// Mitsubishi GX Works2 project: PLC 특수기능 (BKRST)   PLC: Q03UDV

PROGRAM MAIN
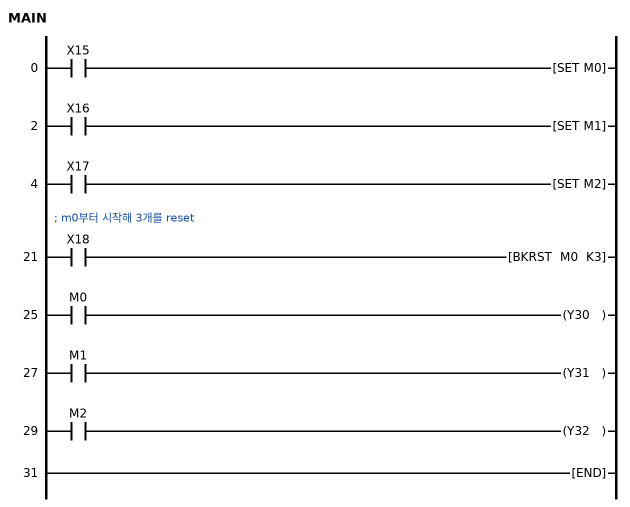
0     LD      X15
      SET     M0
2     LD      X16
      SET     M1
4     LD      X17
      SET     M2
; m0부터 시작해 3개를 reset
21    LD      X18
      BKRST   M0 K3
25    LD      M0
      OUT     Y30
27    LD      M1
      OUT     Y31
29    LD      M2
      OUT     Y32
31    END
END_PROGRAM
